// TIA Portal V20 export
// export: Created 2026-07-10T11:12:24.0943625Z, ExportSetting WithDefaults, DisplayName Totally Integrated Automation Portal, DisplayVersion V20, DisplayName TIA Portal Openness, DisplayVersion V20, DisplayName TIA Portal Version Control Interface, DisplayVersion V20, DisplayName STEP 7 Professional, DisplayVersion V20, DisplayName STEP 7 Safety, DisplayVersion V20, DisplayName WinCC Basic/Comfort/Advanced, DisplayVersion V20, DisplayName WinCC Unified, DisplayVersion V20
FUNCTION_BLOCK "Dampers"   // FB15, SCL
{ S7_Optimized_Access := 'TRUE' }
VERSION : 0.1
// stored: AutoNumber true, IsIECCheckEnabled false, IsRetainMemResEnabled false, MemoryReserve 100, SetENOAutomatically false, UDAEnableTagReadback false
   VAR
      DamperController1 { S7_SetPoint := 'True'} : "DamperController";
      DamperController2 { S7_SetPoint := 'True'} : "DamperController";
      DamperController3 { S7_SetPoint := 'True'} : "DamperController";
   END_VAR
BEGIN
   IF "Inputs_DB".ErrorRCV1 THEN
       #DamperController1.ManualMode := TRUE;
       #DamperController1.ManaulOpen := FALSE;
       #DamperController1.ManualClose := TRUE;
   ELSE
       #DamperController1.ManualMode := "MB".Table.HMI_ManualModeOn;
       #DamperController1.ManaulOpen := "MB".Table.HMI_ManualOpenDamper1;
       #DamperController1.ManualClose := NOT "MB".Table.HMI_ManualOpenDamper1;
   END_IF;

   #DamperController1(TankLevel:="MB".Table.RCV1LevelValue,
                      TankLevelSetpoint:=("MB".Table.LevelRCV1Min + ("MB".Table.LevelRCV1Max-"MB".Table.LevelRCV1Min)/2),
                      TankLevelMin:="MB".Table.LevelRCV1Min,
                      TankLevelMax:="MB".Table.LevelRCV1Max,
                      UsePID:="MB".Table.UsePID,
                      PID_DeadZone:="MB".Table.Damper1_PID_SetpointDeadZone,
                      PID_KP:="MB".Table.Damper1_PID_KP,
                      PID_KI:="MB".Table.Damper1_PID_KI,
                      PID_KD:="MB".Table.Damper1_PID_KD,
                      PID_TI:="MB".Table.Damper1_PID_TI,
                      LimitSwitch0:="RunClose1",
                      LimitSwitch100:="RunOpen1",
                      PouseMove:=5,
                      PositionDeadzone:="MB".Table.Damper1_PositionDeadZone,
                      StartAjustment:="Config".HMI_StartAdjustDamper1,
                      CancelAjustment:="Config".HMI_StopAdjustDamper1,
                      ResetPosition:="Config".HMI_ResetPositionDamper1,
                      Open=>"OutOpen1",
                      Close=>"OutClose1",
                      FullMovingTime:="MB".Table.Damper1_FullMovingTime,
                      SwitchAutoMode := "Damper1_AutoMode");

   "MB".Table."Damper1_Manual/Auto" := "Damper1_AutoMode";

   "MB".Table.Damper1_Position := #DamperController1.CurrentPosition;
   "MB".Table.Damper1_PositionSetpoint := #DamperController1.PositionSetPoint;
   "MB".Table.Damper1_PID_Setpoint := #DamperController1.TankLevelSetpoint;
   "MB".Table.Damper1_AdjustBusy := #DamperController1.AdjustBusy;
   "MB".Table.Damper1_AdjustError := #DamperController1.AdjustError;
   "MB".Table.Damper1_AdjustDone := WORD_TO_BOOL(#DamperController1.AdjustmentDone);

   IF "MB".Table.Damper1_Position > 0 THEN
       "MB".Table."Damper1_Close/Open" := TRUE;
   ELSE
       "MB".Table."Damper1_Close/Open" := FALSE;
   END_IF;

   IF "Inputs_DB".ErrorRCV2 THEN
       #DamperController2.ManualMode := TRUE;
       #DamperController2.ManaulOpen := FALSE;
       #DamperController2.ManualClose := TRUE;
   ELSE
       #DamperController2.ManualMode := "MB".Table.HMI_ManualModeOn;
       #DamperController2.ManaulOpen := "MB".Table.HMI_ManualOpenDamper2;
       #DamperController2.ManualClose := NOT "MB".Table.HMI_ManualOpenDamper2;
   END_IF;

   #DamperController2(TankLevel := "MB".Table.RCV2LevelValue,
                      TankLevelSetpoint := ("MB".Table.LevelRCV2Min + ("MB".Table.LevelRCV2Max - "MB".Table.LevelRCV2Min) / 2),
                      TankLevelMin := "MB".Table.LevelRCV2Min,
                      TankLevelMax := "MB".Table.LevelRCV2Max,
                      UsePID := "MB".Table.UsePID,
                      PID_DeadZone := "MB".Table.Damper2_PID_SetpointDeadZone,
                      PID_KP := "MB".Table.Damper2_PID_KP,
                      PID_KI := "MB".Table.Damper2_PID_KI,
                      PID_KD := "MB".Table.Damper2_PID_KD,
                      PID_TI := "MB".Table.Damper2_PID_TI,
                      LimitSwitch0 := "RunClose2",
                      LimitSwitch100 := "RunOpen2",
                      PouseMove := 5,
                      PositionDeadzone := "MB".Table.Damper2_PositionDeadZone,
                      StartAjustment := "Config".HMI_StartAdjustDamper2,
                      CancelAjustment := "Config".HMI_StopAdjustDamper2,
                      ResetPosition := "Config".HMI_ResetPositionDamper2,
                      Open => "OutOpen2",
                      Close => "OutClose2",
                      FullMovingTime := "MB".Table.Damper2_FullMovingTime,
                      SwitchAutoMode := "Damper2_AutoMode");

   "MB".Table.Damper2_Position := #DamperController2.CurrentPosition;
   "MB".Table.Damper2_PositionSetpoint := #DamperController2.PositionSetPoint;
   "MB".Table.Damper2_PID_Setpoint := #DamperController2.TankLevelSetpoint;
   "MB".Table.Damper2_AdjustBusy := #DamperController2.AdjustBusy;
   "MB".Table.Damper2_AdjustError := #DamperController2.AdjustError;
   "MB".Table.Damper2_AdjustDone := WORD_TO_BOOL(#DamperController2.AdjustmentDone);

   "MB".Table."Damper2_Manual/Auto" := "Damper2_AutoMode";

   #DamperController3(TankLevel := "MB".Table.RCV1LevelValue,
                      TankLevelMin := "MB".Table.LevelRCV1Min,
                      TankLevelMax := "MB".Table.LevelRCV1Max,
                      UsePID := FALSE,
                      LimitSwitch0 := "RunClose1",
                      LimitSwitch100 := "RunOpen1",
                      PouseMove := 5,
                      PositionDeadzone := "MB".Table.Damper1_PositionDeadZone,
                      Open => "OsmosOut",
                      FullMovingTime := "MB".Table.Damper1_FullMovingTime,
                      SwitchAutoMode := TRUE);



   IF "MB".Table.RCV1LevelValue < "MB".Table.LevelRCV1Min THEN
       "OsmosAO" := 5520;
   ELSIF "MB".Table.RCV1LevelValue > "MB".Table.LevelRCV1Max THEN
       "OsmosAO" := 27648;
   ELSE
       "OsmosAO" := REAL_TO_INT(("MB".Table.RCV1LevelValue - "MB".Table.LevelRCV1Min) / ("MB".Table.LevelRCV1Max - "MB".Table.LevelRCV1Min) * (27648 - 5520) + 5520);
   END_IF;

   IF "Inputs_DB".ErrorRCV2 THEN
       #DamperController3.ManualMode := TRUE;
       #DamperController3.ManaulOpen := FALSE;
       #DamperController3.ManualClose := TRUE;
   END_IF;



   IF "MB".Table.Damper2_Position > 0 THEN
       "MB".Table."Damper2_Close/Open" := TRUE;
   ELSE
       "MB".Table."Damper2_Close/Open" := FALSE;
   END_IF;
END_FUNCTION_BLOCK
